FUNCTION_BLOCK RobotControl (* Basic FB with empty ECC *)
  (* Standard: 61499-2 *)
  (* Version 1.0, 2021-09-15, dorofeev *)
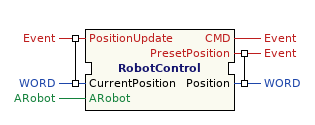
  EVENT_INPUT
    PositionUpdate WITH CurrentPosition;
  END_EVENT
  EVENT_OUTPUT
    CMD;
    PresetPosition WITH Position;
  END_EVENT
  VAR_INPUT
    CurrentPosition : WORD;
  END_VAR
  VAR_OUTPUT
    Position : WORD;
  END_VAR
  SOCKETS
    ARobot : ARobot;
  END_SOCKETS
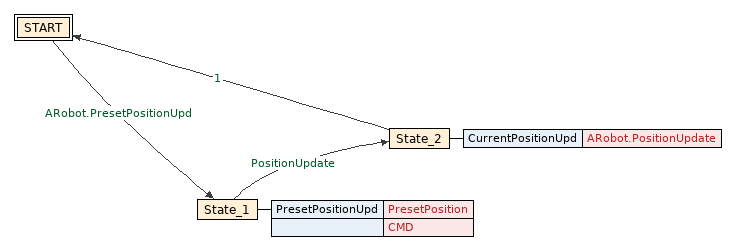
  EC_STATES
    START; (* Initial State *)
    State_1 : PresetPositionUpd -> PresetPosition, -> CMD;
    State_2 : CurrentPositionUpd -> ARobot.PositionUpdate;
  END_STATES
  EC_TRANSITIONS
    State_1 TO State_2 := PositionUpdate;
    START TO State_1 := ARobot.PresetPositionUpd;
    State_2 TO START := 1;
  END_TRANSITIONS
  ALGORITHM PresetPositionUpd IN ST: (* New Algorithm *)
Position := ARobot.PresetPosition;
  END_ALGORITHM
  ALGORITHM CurrentPositionUpd IN ST: (* New Algorithm *)
ARobot.CurrentPosition := CurrentPosition;
  END_ALGORITHM
END_FUNCTION_BLOCK
